FUNCTION_BLOCK AND_COND (* Composite Function Block Type *)
  (* Standard: 61499-2 *)
  (* Version 0.2, 2003-12-05, JHC, Rockwell Automation, Renamed from NEWCOMPFB. *)
  (* Version 0.1, 2002-01-08, JHC, Rockwell Automation, Added DLY FB as example. *)
  (* Version 0.0, 2000-05-27, JHC, Rockwell Automation *)
  (* Compiler header: package fb.rt.student; *)
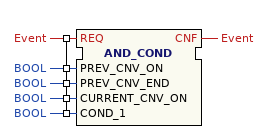
  EVENT_INPUT
    REQ WITH PREV_CNV_ON, PREV_CNV_END, CURRENT_CNV_ON, COND_1; (* Normal Execution Request *)
  END_EVENT
  EVENT_OUTPUT
    CNF; (* Execution Confirmation *)
  END_EVENT
  VAR_INPUT
    PREV_CNV_ON : BOOL;
    PREV_CNV_END : BOOL;
    CURRENT_CNV_ON : BOOL;
    COND_1 : BOOL;
  END_VAR
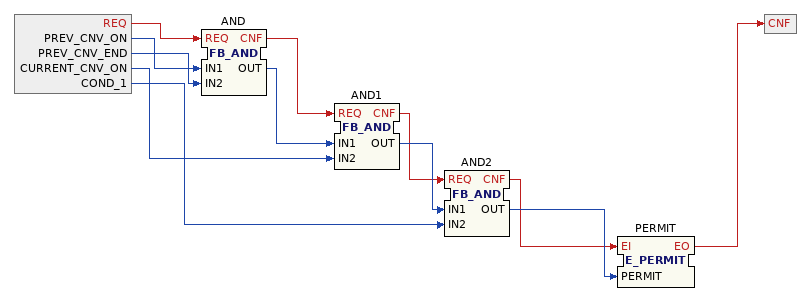
  FBS
    PERMIT : E_PERMIT;
    AND : FB_AND;
    AND1 : FB_AND;
    AND2 : FB_AND;
  END_FBS
  EVENT_CONNECTIONS
    AND.CNF TO AND1.REQ;
    AND1.CNF TO AND2.REQ;
    REQ TO AND.REQ;
    AND2.CNF TO PERMIT.EI;
    PERMIT.EO TO CNF;
  END_CONNECTIONS
  DATA_CONNECTIONS
    PREV_CNV_ON TO AND.IN1;
    PREV_CNV_END TO AND.IN2;
    AND.OUT TO AND1.IN1;
    CURRENT_CNV_ON TO AND1.IN2;
    AND1.OUT TO AND2.IN1;
    COND_1 TO AND2.IN2;
    AND2.OUT TO PERMIT.PERMIT;
  END_CONNECTIONS
END_FUNCTION_BLOCK
